	FUNCTION_BLOCK FB 404
	TITLE =G304M WITHERING AIR KILN 2
	//COPYRIGHT:    (C) 2009  BUHLER AG, CH-9240 UZWIL, SWITZERLAND
	//
	//PRODUCT:      WinCoS_BIW01_09
	//
	//TITLE:        WITHERING AIR KILN 2
	//                Machine group control
	//                Maschinengruppensteuerung
	//
	//--------------------------------------------------------------------------------
	//
	//IDENT:        AUTHOR:             DEPT:                              DATE:
	//
	//P01_FB404.1.0 K.Renz              CSB41                              09.Okt.2009
	//             1st Release
	//
	//--------------------------------------------------------------------------------
	//
	//PURPOSE:
	//
	//MANUAL :
	//
	//RESTRICTIONS:
	//
	//--------------------------------------------------------------------------------
	AUTHOR  : KR
	FAMILY  : USW
	VERSION : 9.9


	VAR
	  Gr       : FB10;	//Standard interface to group
	  InOutValue1    : DINT; //Data for user
	  InOutValue2    : DINT; //Data for user
	  OutWayConflict : BOOL;	//Data for user
	  OutSelectionOk : BOOL;	//Data for user
	  CmdNewValue : BOOL;	//Data for user
	  CmdNewJob   : BOOL;	//Data for user
	  OutCodeOK   : BOOL;	//Data for user
	  InEndOfJob  : BOOL ;	//Data for user
	  staWayOk      : BOOL ;	//Data for user
	  EdgeStartRelease : BOOL ;	//Data for user
	  USW8  : BOOL;	//Data for user
	  USW9 : BOOL;	//Data for user
	  USW10: BOOL;	//Data for user
	  USW11: BOOL;	//Data for user
	  USW12: BOOL;	//Data for user
	  USW13: BOOL;	//Data for user
	  USW14: BOOL;	//Data for user
	  USW15: BOOL;	//Data for user
	     #A_3245_MXZ11 : FB20;   // VLS4Ctrl
	     #A_3245_MXZ11I1 : FB14;   // DigInpCont
	     #A_3245_MXZ11I2 : FB14;   // DigInpCont
	     #A_3246_MXZ11 : FB20;   // VLS4Ctrl
	     #A_3246_MXZ11I1 : FB14;   // DigInpCont
	     #A_3246_MXZ11I2 : FB14;   // DigInpCont
	     #A_3245_BZS14 : FB14;   // DigInpCont
	     #A_3245_BZS15 : FB14;   // DigInpCont
	     #A_3246_BZS14 : FB14;   // DigInpCont
	     #A_3246_BZS15 : FB14;   // DigInpCont
	END_VAR
	VAR_TEMP
	   tmpEnable		: BOOL;
	   tmpFlag  		: BOOL;
	   tmpCmdNext		: BOOL;
	   tmpLocal  		: BOOL;
	   tmpAspOk  		: BOOL;
	   tmpHWStop 		: BOOL;
	   tmpInstanzDBNo       : INT ;
	END_VAR
	BEGIN
	NETWORK
	TITLE =
	NETWORK
	TITLE =Read command from group control
	//Parameter
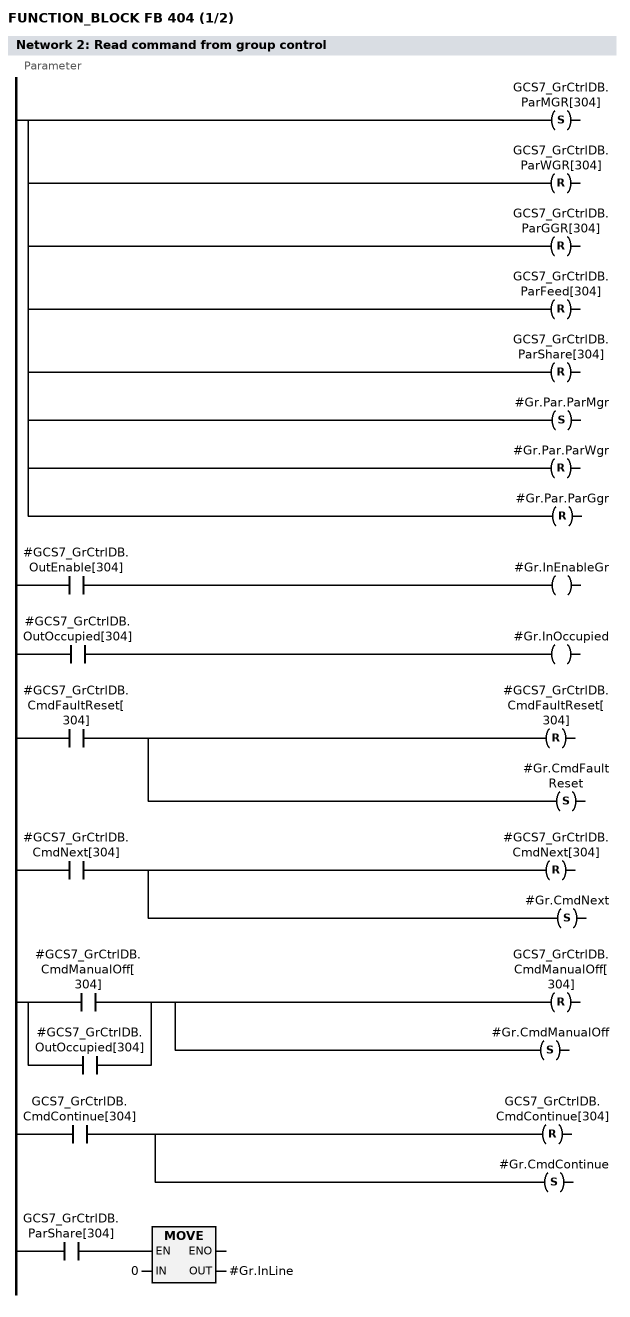
	      SET;
	      S   GCS7_GrCtrlDB.ParMGR[304];
	      R   GCS7_GrCtrlDB.ParWGR[304];
	      R   GCS7_GrCtrlDB.ParGGR[304];
	      R   GCS7_GrCtrlDB.ParFeed[304];
	      R   GCS7_GrCtrlDB.ParShare[304];
	      S   #Gr.Par.ParMgr;
	      R   #Gr.Par.ParWgr;
	      R   #Gr.Par.ParGgr;
	//Command
	      U   #GCS7_GrCtrlDB.OutEnable[304];
	      =   #Gr.InEnableGr;
	      U   #GCS7_GrCtrlDB.OutOccupied[304];
	      =   #Gr.InOccupied;
	      U   #GCS7_GrCtrlDB.CmdFaultReset[304];
	      R   #GCS7_GrCtrlDB.CmdFaultReset[304];
	      S   #Gr.CmdFaultReset;
	      U  #GCS7_GrCtrlDB.CmdNext[304];
	      R   #GCS7_GrCtrlDB.CmdNext[304];
	      S   #Gr.CmdNext;
	      U   #GCS7_GrCtrlDB.CmdManualOff[304];
	      O   #GCS7_GrCtrlDB.OutOccupied[304];
	      R   GCS7_GrCtrlDB.CmdManualOff[304];
	      S   #Gr.CmdManualOff;
	      U  GCS7_GrCtrlDB.CmdContinue[304];
	      R   GCS7_GrCtrlDB.CmdContinue[304];
	      S   #Gr.CmdContinue;
	//Init Line Number
	      U   GCS7_GrCtrlDB.ParShare[304];
	      SPBN WE00;
	      L     0;
	      T     #Gr.InLine;
	WE00: NOP   0;
	NETWORK
	TITLE =Call Methode Control
	// 1. Handle Interface PCControl
	// 2. Prepare mode --> ModePassive,ModeActive,ModeIdling
	// 3. Reset global flags of the group
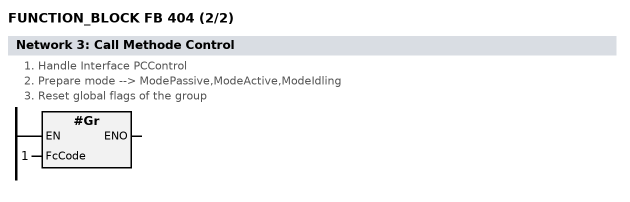
	      CALL #Gr (
	           FcCode                   := 1);
	NETWORK
	TITLE =Restart Idling Time
		L  #Gr.Par.ParIdling;
		L  2;
		>=I;
		SPB IdTm;
		T  #Gr.Par.ParIdling;
	IdTm:   NOP 0;
	      CLR;
	      S    #Gr.CmdRestartIdling;
	NETWORK
	TITLE =Prepare global flags
	NETWORK
	TITLE =Set Pattern (Target position)
	NETWORK
	TITLE =Interlocking WayOk
	//
	NETWORK
	TITLE =Interlocking Autostart
		CLR;
		R   #Gr.OutAutostart;
	NETWORK
	TITLE =Interlocking Enable
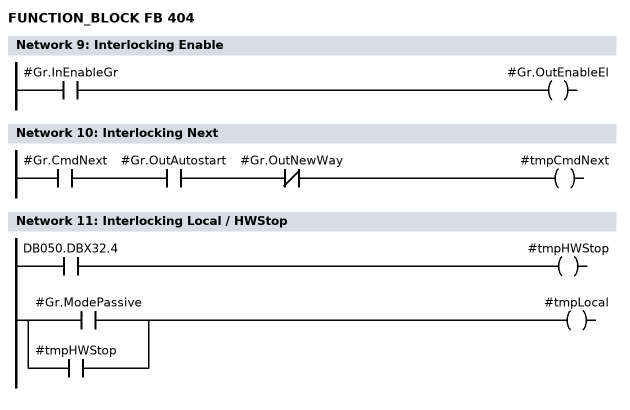
	      U     #Gr.InEnableGr;
	      =     #Gr.OutEnableEl;

	NETWORK
	TITLE =Interlocking Next
	      U     #Gr.CmdNext;
	      U     #Gr.OutAutostart;
	      UN    #Gr.OutNewWay;
	      =    #tmpCmdNext;

	NETWORK
	TITLE =Interlocking Local / HWStop
	      U    DB050.DBX32.4;
	      =    #tmpHWStop;

	      U    #Gr.ModePassive;
	      O    #tmpHWStop;
	      =    #tmpLocal;

	NETWORK
	TITLE ==A-3245-MXZ11 : LOUVER WITHERING AIR 1
	NOP 0;
	//-InLocal---
	      U     #tmpLocal;
	      =     #A_3245_MXZ11.InLocal;
	//
	//-Interlocking---
	      UN     #Gr.OutEnableEl;
	      =     #A_3245_MXZ11.InLN;
	      U    #Gr.OutEnableEl;
	      S     #A_3245_MXZ11.CmdMiddle1;
	      S     #A_3245_MXZ11.CmdMiddle2;
	      S     #A_3245_MXZ11.CmdHN;
	//
	//-Read inputs---
	      U     E 1002.0;
	      =     #A_3245_MXZ11.InpLN;
	      CLR;
	      =     #A_3245_MXZ11.InpMiddle1;
	      U     E 1002.1;
	      =     #A_3245_MXZ11.InpHN;
	      U   DB050.DBX32.4;
	      =     #A_3245_MXZ11.InHWStop;
	       U     PLC_DPInfo.Master[1].SlavesError[101];
	       =       #A_3245_MXZ11.InDPFault;
	//
	//-Set Parameters---
	//
	//-Call object control---
	      CALL  #A_3245_MXZ11;
	//
	//-Write outputs---
	      U     #A_3245_MXZ11.OutpLN;
	      =     A 1002.0;
	      U     #A_3245_MXZ11.OutpHN;
	      =     A 1002.1;
	NETWORK
	TITLE ==A-3245-MXZ11I1 : LOUVER WITHERING AIR 1 CLOSING
	NOP 0;
	//-InLocal---
	      U     #tmpLocal;
	      =     #A_3245_MXZ11I1.InLocal;
	//
	//-Monitoring---
	      SET;
	      =      #A_3245_MXZ11I1.InMonTrue;
	      CLR;
	      =      #A_3245_MXZ11I1.InMonFalse;
	//
	//-PreAlarm---
	      CLR;
	      =      #A_3245_MXZ11I1.InPreAlarmTrue;
	      CLR;
	      =      #A_3245_MXZ11I1.InPreAlarmFalse;
	//
	//-Additional commands---
	//      CLR
	//      S     #A_3245_MXZ11I1.CmdRunTimeOutTime
	//
	//-Read inputs---
	      U     E 1002.0;
	      =     #A_3245_MXZ11I1.InpTrue;
	      U   DB050.DBX32.4;
	      =     #A_3245_MXZ11I1.InHWStop;
	       U     PLC_DPInfo.Master[1].SlavesError[101];
	       =       #A_3245_MXZ11I1.InDPFault;
	//
	//-Set Parameters---
	//
	//-Call object control---
	      CALL  #A_3245_MXZ11I1;
	//
	//-Write outputs---
	NETWORK
	TITLE ==A-3245-MXZ11I2 : LOUVER WITHERING AIR 1 OPENING
	NOP 0;
	//-InLocal---
	      U     #tmpLocal;
	      =     #A_3245_MXZ11I2.InLocal;
	//
	//-Monitoring---
	      SET;
	      =      #A_3245_MXZ11I2.InMonTrue;
	      CLR;
	      =      #A_3245_MXZ11I2.InMonFalse;
	//
	//-PreAlarm---
	      CLR;
	      =      #A_3245_MXZ11I2.InPreAlarmTrue;
	      CLR;
	      =      #A_3245_MXZ11I2.InPreAlarmFalse;
	//
	//-Additional commands---
	//      CLR
	//      S     #A_3245_MXZ11I2.CmdRunTimeOutTime
	//
	//-Read inputs---
	      U     E 1002.1;
	      =     #A_3245_MXZ11I2.InpTrue;
	      U   DB050.DBX32.4;
	      =     #A_3245_MXZ11I2.InHWStop;
	       U     PLC_DPInfo.Master[1].SlavesError[101];
	       =       #A_3245_MXZ11I2.InDPFault;
	//
	//-Set Parameters---
	//
	//-Call object control---
	      CALL  #A_3245_MXZ11I2;
	//
	//-Write outputs---
	NETWORK
	TITLE ==A-3246-MXZ11 : LOUVER WITHERING AIR 2
	NOP 0;
	//-InLocal---
	      U     #tmpLocal;
	      =     #A_3246_MXZ11.InLocal;
	//
	//-Interlocking---
	      UN     #Gr.OutEnableEl;
	      =     #A_3246_MXZ11.InLN;
	      U    #Gr.OutEnableEl;
	      S     #A_3246_MXZ11.CmdMiddle1;
	      S     #A_3246_MXZ11.CmdMiddle2;
	      S     #A_3246_MXZ11.CmdHN;
	//
	//-Read inputs---
	      U     E 1002.2;
	      =     #A_3246_MXZ11.InpLN;
	      CLR;
	      =     #A_3246_MXZ11.InpMiddle1;
	      U     E 1002.3;
	      =     #A_3246_MXZ11.InpHN;
	      U   DB050.DBX32.4;
	      =     #A_3246_MXZ11.InHWStop;
	       U     PLC_DPInfo.Master[1].SlavesError[101];
	       =       #A_3246_MXZ11.InDPFault;
	//
	//-Set Parameters---
	//
	//-Call object control---
	      CALL  #A_3246_MXZ11;
	//
	//-Write outputs---
	      U     #A_3246_MXZ11.OutpLN;
	      =     A 1002.2;
	      U     #A_3246_MXZ11.OutpHN;
	      =     A 1002.3;
	NETWORK
	TITLE ==A-3246-MXZ11I1 : LOUVER WITHERING AIR 2 CLOSING
	NOP 0;
	//-InLocal---
	      U     #tmpLocal;
	      =     #A_3246_MXZ11I1.InLocal;
	//
	//-Monitoring---
	      SET;
	      =      #A_3246_MXZ11I1.InMonTrue;
	      CLR;
	      =      #A_3246_MXZ11I1.InMonFalse;
	//
	//-PreAlarm---
	      CLR;
	      =      #A_3246_MXZ11I1.InPreAlarmTrue;
	      CLR;
	      =      #A_3246_MXZ11I1.InPreAlarmFalse;
	//
	//-Additional commands---
	//      CLR
	//      S     #A_3246_MXZ11I1.CmdRunTimeOutTime
	//
	//-Read inputs---
	      U     E 1002.2;
	      =     #A_3246_MXZ11I1.InpTrue;
	      U   DB050.DBX32.4;
	      =     #A_3246_MXZ11I1.InHWStop;
	       U     PLC_DPInfo.Master[1].SlavesError[101];
	       =       #A_3246_MXZ11I1.InDPFault;
	//
	//-Set Parameters---
	//
	//-Call object control---
	      CALL  #A_3246_MXZ11I1;
	//
	//-Write outputs---
	NETWORK
	TITLE ==A-3246-MXZ11I2 : LOUVER WITHERING AIR 2 OPENING
	NOP 0;
	//-InLocal---
	      U     #tmpLocal;
	      =     #A_3246_MXZ11I2.InLocal;
	//
	//-Monitoring---
	      SET;
	      =      #A_3246_MXZ11I2.InMonTrue;
	      CLR;
	      =      #A_3246_MXZ11I2.InMonFalse;
	//
	//-PreAlarm---
	      CLR;
	      =      #A_3246_MXZ11I2.InPreAlarmTrue;
	      CLR;
	      =      #A_3246_MXZ11I2.InPreAlarmFalse;
	//
	//-Additional commands---
	//      CLR
	//      S     #A_3246_MXZ11I2.CmdRunTimeOutTime
	//
	//-Read inputs---
	      U     E 1002.3;
	      =     #A_3246_MXZ11I2.InpTrue;
	      U   DB050.DBX32.4;
	      =     #A_3246_MXZ11I2.InHWStop;
	       U     PLC_DPInfo.Master[1].SlavesError[101];
	       =       #A_3246_MXZ11I2.InDPFault;
	//
	//-Set Parameters---
	//
	//-Call object control---
	      CALL  #A_3246_MXZ11I2;
	//
	//-Write outputs---
	NETWORK
	TITLE ==A-3245-BZS14 : LOUVER WITHERING AIR 1 CLOSED
	NOP 0;
	//-InLocal---
	      U     #tmpLocal;
	      =     #A_3245_BZS14.InLocal;
	//
	//-Monitoring---
	      CLR;
	      =      #A_3245_BZS14.InMonTrue;
	      CLR;
	      =      #A_3245_BZS14.InMonFalse;
	//
	//-PreAlarm---
	      CLR;
	      =      #A_3245_BZS14.InPreAlarmTrue;
	      CLR;
	      =      #A_3245_BZS14.InPreAlarmFalse;
	//
	//-Additional commands---
	//      CLR
	//      S     #A_3245_BZS14.CmdRunTimeOutTime
	//
	//-Read inputs---
	      U     E 1005.6;
	      =     #A_3245_BZS14.InpTrue;
	      U   DB050.DBX32.4;
	      =     #A_3245_BZS14.InHWStop;
	       U     PLC_DPInfo.Master[1].SlavesError[101];
	       =       #A_3245_BZS14.InDPFault;
	//
	//-Set Parameters---
	//
	//-Call object control---
	      CALL  #A_3245_BZS14;
	//
	//-Write outputs---
	NETWORK
	TITLE ==A-3245-BZS15 : LOUVER WITHERING AIR 1 OPENED
	NOP 0;
	//-InLocal---
	      U     #tmpLocal;
	      =     #A_3245_BZS15.InLocal;
	//
	//-Monitoring---
	      CLR;
	      =      #A_3245_BZS15.InMonTrue;
	      CLR;
	      =      #A_3245_BZS15.InMonFalse;
	//
	//-PreAlarm---
	      CLR;
	      =      #A_3245_BZS15.InPreAlarmTrue;
	      CLR;
	      =      #A_3245_BZS15.InPreAlarmFalse;
	//
	//-Additional commands---
	//      CLR
	//      S     #A_3245_BZS15.CmdRunTimeOutTime
	//
	//-Read inputs---
	      U     E 1005.7;
	      =     #A_3245_BZS15.InpTrue;
	      U   DB050.DBX32.4;
	      =     #A_3245_BZS15.InHWStop;
	       U     PLC_DPInfo.Master[1].SlavesError[101];
	       =       #A_3245_BZS15.InDPFault;
	//
	//-Set Parameters---
	//
	//-Call object control---
	      CALL  #A_3245_BZS15;
	//
	//-Write outputs---
	NETWORK
	TITLE ==A-3246-BZS14 : LOUVER WITHERING AIR 2 CLOSED
	NOP 0;
	//-InLocal---
	      U     #tmpLocal;
	      =     #A_3246_BZS14.InLocal;
	//
	//-Monitoring---
	      CLR;
	      =      #A_3246_BZS14.InMonTrue;
	      CLR;
	      =      #A_3246_BZS14.InMonFalse;
	//
	//-PreAlarm---
	      CLR;
	      =      #A_3246_BZS14.InPreAlarmTrue;
	      CLR;
	      =      #A_3246_BZS14.InPreAlarmFalse;
	//
	//-Additional commands---
	//      CLR
	//      S     #A_3246_BZS14.CmdRunTimeOutTime
	//
	//-Read inputs---
	      U     E 1006.0;
	      =     #A_3246_BZS14.InpTrue;
	      U   DB050.DBX32.4;
	      =     #A_3246_BZS14.InHWStop;
	       U     PLC_DPInfo.Master[1].SlavesError[101];
	       =       #A_3246_BZS14.InDPFault;
	//
	//-Set Parameters---
	//
	//-Call object control---
	      CALL  #A_3246_BZS14;
	//
	//-Write outputs---
	NETWORK
	TITLE ==A-3246-BZS15 : LOUVER WITHERING AIR 2 OPENED
	NOP 0;
	//-InLocal---
	      U     #tmpLocal;
	      =     #A_3246_BZS15.InLocal;
	//
	//-Monitoring---
	      CLR;
	      =      #A_3246_BZS15.InMonTrue;
	      CLR;
	      =      #A_3246_BZS15.InMonFalse;
	//
	//-PreAlarm---
	      CLR;
	      =      #A_3246_BZS15.InPreAlarmTrue;
	      CLR;
	      =      #A_3246_BZS15.InPreAlarmFalse;
	//
	//-Additional commands---
	//      CLR
	//      S     #A_3246_BZS15.CmdRunTimeOutTime
	//
	//-Read inputs---
	      U     E 1006.1;
	      =     #A_3246_BZS15.InpTrue;
	      U   DB050.DBX32.4;
	      =     #A_3246_BZS15.InHWStop;
	       U     PLC_DPInfo.Master[1].SlavesError[101];
	       =       #A_3246_BZS15.InDPFault;
	//
	//-Set Parameters---
	//
	//-Call object control---
	      CALL  #A_3246_BZS15;
	//
	//-Write outputs---
	NETWORK
	TITLE =Test Fault
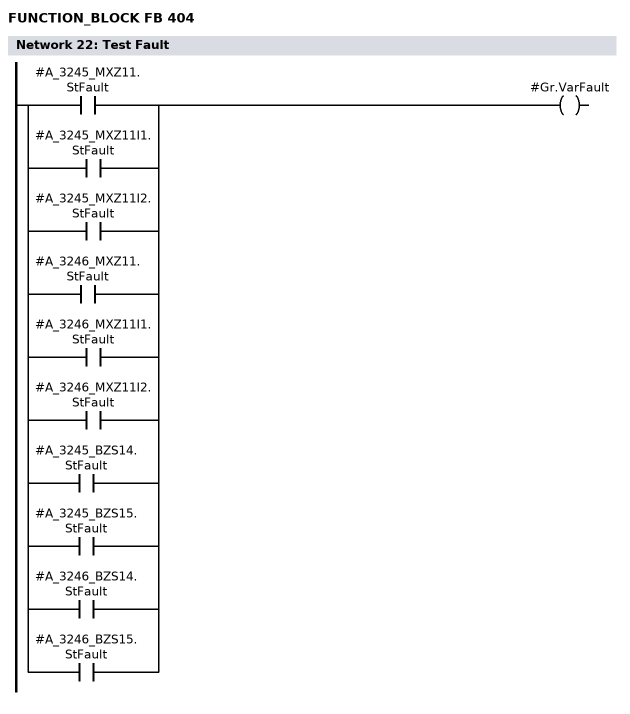
	      U     #A_3245_MXZ11.StFault;
	      O     #A_3245_MXZ11I1.StFault;
	      O     #A_3245_MXZ11I2.StFault;
	      O     #A_3246_MXZ11.StFault;
	      O     #A_3246_MXZ11I1.StFault;
	      O     #A_3246_MXZ11I2.StFault;
	      O     #A_3245_BZS14.StFault;
	      O     #A_3245_BZS15.StFault;
	      O     #A_3246_BZS14.StFault;
	      O     #A_3246_BZS15.StFault;
	      =     #Gr.VarFault;
	NETWORK
	TITLE =Test Warning
	      CLR;
	      =     #Gr.OutWarning;
	NETWORK
	TITLE =Test Stopped
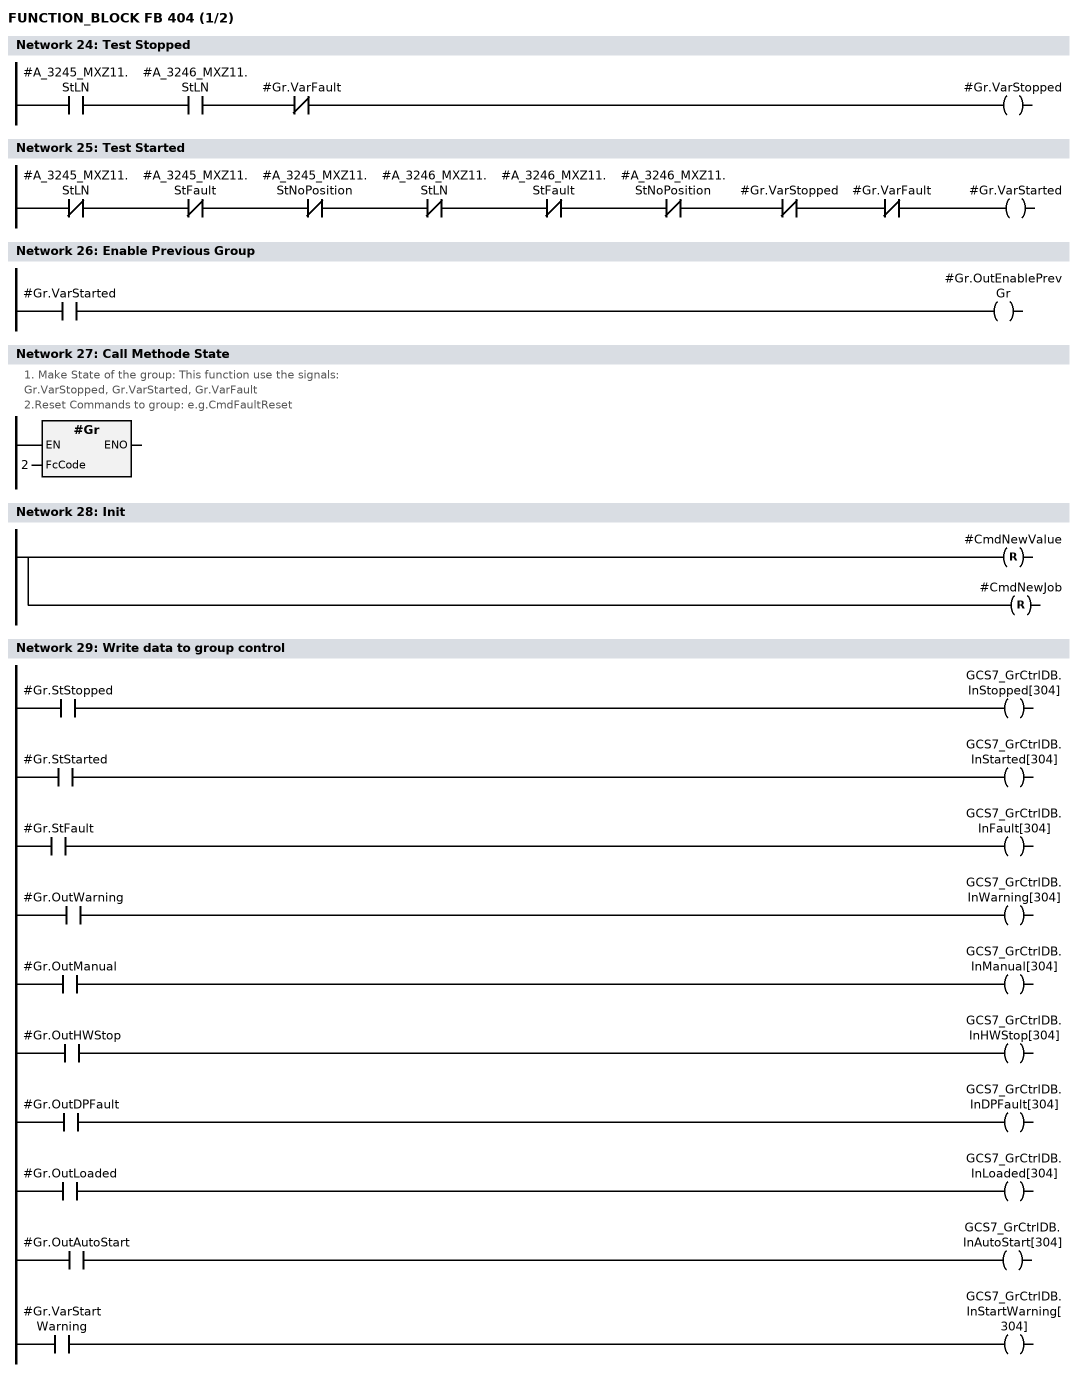
	      U     #A_3245_MXZ11.StLN;
	      U     #A_3246_MXZ11.StLN;
	      UN   #Gr.VarFault;
	      =     #Gr.VarStopped;
	NETWORK
	TITLE =Test Started
	      UN     #A_3245_MXZ11.StLN;
	      UN     #A_3245_MXZ11.StFault;
	      UN     #A_3245_MXZ11.StNoPosition;
	      UN     #A_3246_MXZ11.StLN;
	      UN     #A_3246_MXZ11.StFault;
	      UN     #A_3246_MXZ11.StNoPosition;
	      UN  #Gr.VarStopped;
	      UN  #Gr.VarFault;
	      =     #Gr.VarStarted;
	NETWORK
	TITLE =Enable Previous Group
	      U    #Gr.VarStarted;
	      =     #Gr.OutEnablePrevGr;
	NETWORK
	TITLE =Call Methode State
	//1. Make State of the group: This function use the signals:
	//        Gr.VarStopped, Gr.VarStarted, Gr.VarFault
	//2.Reset Commands to group: e.g.CmdFaultReset
	      CALL #Gr (
	           FcCode                   := 2);
	NETWORK
	TITLE =Init
	      SET;
	      R    #CmdNewValue;
	      R    #CmdNewJob;
	NETWORK
	TITLE =Write data to group control
	      U   #Gr.StStopped;
	      =   GCS7_GrCtrlDB.InStopped[304];
	      U   #Gr.StStarted;
	      =   GCS7_GrCtrlDB.InStarted[304];
	      U   #Gr.StFault;
	      =   GCS7_GrCtrlDB.InFault[304];
	      U   #Gr.OutWarning;
	      =   GCS7_GrCtrlDB.InWarning[304];
	      U   #Gr.OutManual;
	      =   GCS7_GrCtrlDB.InManual[304];
	      U   #Gr.OutHWStop;
	      =   GCS7_GrCtrlDB.InHWStop[304];
	      U   #Gr.OutDPFault;
	      =   GCS7_GrCtrlDB.InDPFault[304];
	      U   #Gr.OutLoaded;
	      =   GCS7_GrCtrlDB.InLoaded[304];
	      U   #Gr.OutAutoStart;
	      =   GCS7_GrCtrlDB.InAutoStart[304];
	      U   #Gr.VarStartWarning;
	      =   GCS7_GrCtrlDB.InStartWarning[304];
	NETWORK
	TITLE =End of block
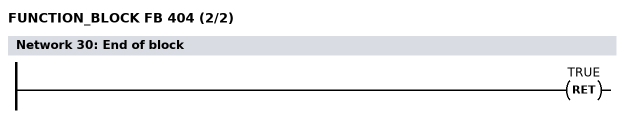

	BE

	END_FUNCTION_BLOCK
